// TIA Portal project "BK_Proje_Odevi_6_Video1" (V15.1)
// Vorlageprojekt für das Buch mit Zielsystem S7-1200

(* hardware
DEVICE "S7-1200-Station_1"  S7-1200 Station
   slot 0: "Baugruppenträger_0"  Rack  V1.0
   slot 1: "PLC_1"  CPU 1211C DC/DC/DC  6ES7 211-1AE40-0XB0  V4.1
*)

// ===== PLC "PLC_1"  CPU 1211C DC/DC/DC =====

VAR_GLOBAL   // PLC tag table "Standard-Variablentabelle"
   "Tag_1" AT %A0.0 : Bool;
   "Tag_2" AT %E0.0 : Bool;
   "Tag_3" AT %E0.1 : Bool;
   "Tag_4" AT %ID30 : Real;
   "Tag_5" AT %MD30 : Real;
   "Tag_6" AT %QD38 : DInt;
   "Tag_7" AT %QD30 : Real;
   "Tag_8" AT %QD34 : Real;
   "Tag_9" AT %ID34 : Real;
END_VAR

FUNCTION "Olceklendirme" : Void   // FC1, SCL
{ S7_Optimized_Access := 'TRUE' }
VERSION : 0.1
   VAR_INPUT
      Seviye_Sensoru : Real;
   END_VAR
   VAR_OUTPUT
      Olcekli_Sensor : Real;   // Yuzde bazında
      Olcekli_Yukseklik : DInt;   // Cm bazında
   END_VAR
   VAR_TEMP
      Olcekli_Yukseklik_Real : Real;   // Donusturme icin
   END_VAR
BEGIN
   //Aralıgı 0.0 - 10.0'dan 0-100%'a donusturme
   #Olcekli_Sensor := #Seviye_Sensoru * 10.0;

   //Aralıgı 0.0 - 10.0'dan 0-300cm'ye donustume
   #Olcekli_Yukseklik_Real:= #Seviye_Sensoru* 30.0;
   #Olcekli_Yukseklik := REAL_TO_INT(#Olcekli_Yukseklik_Real);
END_FUNCTION

FUNCTION "ON/OFF_ile_Otomasyon_Kontrol" : Void   // FC2, SCL
{ S7_Optimized_Access := 'TRUE' }
VERSION : 0.1
   VAR_INPUT
      Seviye_Yuzde_Deger : Real;
      Bosaltma_Butonu : Bool;
   END_VAR
   VAR_OUTPUT
      Doldurma_Vanasi : Real;
      Bosaltma_Vanasi : Real;
   END_VAR
BEGIN
   //Eger (IF) tank seviyesi < 40% = doldurma vanasini 100% ac
   //Eger (IF) tank seviyesi > 40% ve (AND) tank seviyesi < 80% = doldurma vanasini 50% ac
   //Eger (IF) tank seviyesi > 80% = doldurma vanasini 0% ac
   IF #Seviye_Yuzde_Deger < 40.0 THEN

       #Doldurma_Vanasi := 10.0; // Statement section IF

   ELSIF #Seviye_Yuzde_Deger > 40.0 AND #Seviye_Yuzde_Deger < 80.0 THEN

       #Doldurma_Vanasi := 5.0; // Statement section ELSIF

   ELSIF #Seviye_Yuzde_Deger > 80.0 THEN

       #Doldurma_Vanasi := 0.0;// Statement section ELSE

   END_IF;

   //Use Toggle button TO drain the level (at 50% flow rate)
   IF #Bosaltma_Butonu = 1 THEN

       #Bosaltma_Vanasi := 5.0;

   END_IF;
END_FUNCTION

FUNCTION "Orantisal_Kontrol" : Void   // FC3, SCL
{ S7_Optimized_Access := 'TRUE' }
VERSION : 0.1
   VAR_INPUT
      Ayar_Kontrol : Real;
      Seviye_Sensoru : Real;
      Kp : Real;   // Potansiyometredeki Orantisal Kazanc
   END_VAR
   VAR_OUTPUT
      Bosaltma_Vanasi : Real;
      Doldurma_Vanasi : Real;
   END_VAR
   VAR_TEMP
      Hata : Real;   // Fark
      u : Real;   // Orantisal Kontrol Cikisi
   END_VAR
BEGIN
   //Hata:
   #Hata:= #Ayar_Kontrol - #Seviye_Sensoru;

   //Orantisal Kontrol:
   #u := #Hata * #Kp;

   //Cikis:
   #Doldurma_Vanasi := #u; //Ornegin Ayar_Kontrol = 75% ve Seviye 50% iken.
   #Bosaltma_Vanasi := - #u; //Ornegin Ayar_Kontrol = 50% ve Seviye 100% iken.
END_FUNCTION

FUNCTION "MHJ-PLC-Lab-Function-S71200" : Void   // FC9000, SCL
{ S7_Optimized_Access := 'TRUE' }
VERSION : 0.1
   VAR_TEMP
      rdTimeReturn : Int;
      outputTime : DTL;
      SyncVal : Byte;
      forVal : Int;
      forVal_2 : Int;
      Value : Byte;
   END_VAR
   VAR CONSTANT
      CompVal : Byte := 16#34;
      Value_01 : Byte := 16#11;
      Value_01_DW : DWord := 16#A165_D992;
      Value_02_DW : DWord := 16#58BE_4401;
   END_VAR
BEGIN

   #Value:=PEEK(area := 16#82,
        dbNumber := 0,
        byteOffset := 511);
   #Value := #Value + 1;

   POKE(area := 16#82,
        dbNumber := 0,
        byteOffset := 511,
        value := #Value);

   POKE(area:=16#81,
        dbNumber:=0,
        byteOffset:=1016,
        value:=#Value_01_DW);
   POKE(area := 16#81,
        dbNumber := 0,
        byteOffset := 1020,
        value := #Value_02_DW);

   POKE(area := 16#81,
        dbNumber := 0,
        byteOffset := 511,
        value := B#16#00);

   FOR #forVal := 0 TO 120 DO
       FOR #forVal_2:=0 TO 10 DO
           #rdTimeReturn:=RD_SYS_T(#outputTime);
           #rdTimeReturn := WR_SYS_T(#outputTime);
           #rdTimeReturn := RD_SYS_T(#outputTime);
           #rdTimeReturn := WR_SYS_T(#outputTime);
       END_FOR;
       #SyncVal:= PEEK(area := 16#81,
                      dbNumber := 0,
                      byteOffset := 511);
       IF #SyncVal = #CompVal THEN
          GOTO M_1;
       END_IF;
   END_FOR;
   RETURN;

   M_1:
   POKE(area := 16#81,
        dbNumber := 0,
        byteOffset := 511,
        value := B#16#0);
END_FUNCTION

ORGANIZATION_BLOCK "Main"   // OB1, LAD, ProgramCycle
TITLE = "Main Program Sweep (Cycle)"
{ S7_Optimized_Access := 'TRUE' }
VERSION : 0.1
   VAR_INPUT
      Initial_Call : Bool;   // Initial call of this OB
      Remanence : Bool;   // =True, if remanent data are available
   END_VAR
BEGIN

REGION Network 1: Konnektierungsbaustein für PLC-Lab / Programi Factoy IO'ya Uyarlama
   // Im Netzwerk 1 wird der Konnektierungsbaustein für PLC-Lab aufgerufen.
   // Dieser Aufruf darf nicht entfernt werden!
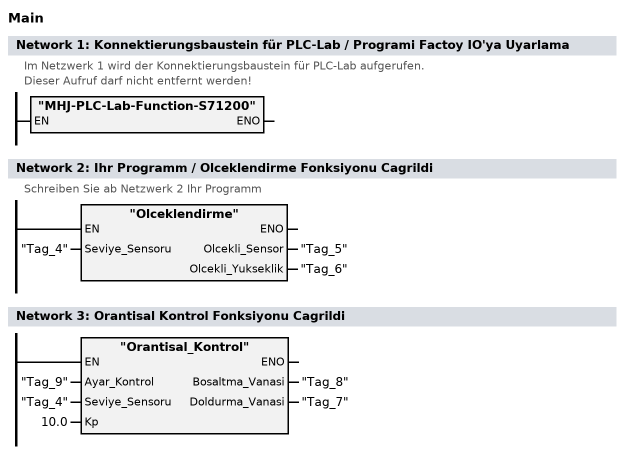
   RUNG wire#powerrail
      "MHJ-PLC-Lab-Function-S71200"()
   END_RUNG
   // the same network as SCL:
   "MHJ-PLC-Lab-Function-S71200"();
END_REGION

REGION Network 2: Ihr Programm / Olceklendirme Fonksiyonu Cagrildi
   // Schreiben Sie ab Netzwerk 2 Ihr Programm
   RUNG wire#powerrail
      "Olceklendirme"(Seviye_Sensoru := "Tag_4", Olcekli_Sensor => "Tag_5", Olcekli_Yukseklik => "Tag_6")
   END_RUNG
   // the same network as SCL:
   "Olceklendirme"(Seviye_Sensoru := "Tag_4", Olcekli_Sensor => "Tag_5", Olcekli_Yukseklik => "Tag_6");
END_REGION

REGION Network 3: Orantisal Kontrol Fonksiyonu Cagrildi
   RUNG wire#powerrail
      "Orantisal_Kontrol"(Ayar_Kontrol := "Tag_9", Seviye_Sensoru := "Tag_4", Kp := 10.0, Bosaltma_Vanasi => "Tag_8", Doldurma_Vanasi => "Tag_7")
   END_RUNG
   // the same network as SCL:
   "Orantisal_Kontrol"(Ayar_Kontrol := "Tag_9",
                       Seviye_Sensoru := "Tag_4",
                       Kp := 10.0,
                       Bosaltma_Vanasi => "Tag_8",
                       Doldurma_Vanasi => "Tag_7");
END_REGION
END_ORGANIZATION_BLOCK